Staubli VAL3: Txt_PkgInit.pgx

program Txt_PkgInit()
begin
  n_sTxt=0
  call Txt_initData()
  call TxtReadRoom1()
  if nTxtTotal>1
    call TxtReadRoom2()
  endIf
  bTxtPrSv=true
  sScrPts="OK"
  call hmi_refreshmain()
end
